// TIA Portal V21 export
DATA_BLOCK "RMAdd"   // DB305
AUTHOR : PRECISE
FAMILY : PRECISE
// stored: AutoNumber false, InstanceOfName FB310, InstanceOfType FB
"FB310"
   // VAR_INPUT
   //    Enable : Bool;
   //    Disable : Bool;
   //    Fault : Bool;
   //    SecPulse : Bool;
   //    AlwaysTrue : Bool;
   //    StartConfirmationPopupSel : Bool;
   //    EndConfirmationPopupSel : Bool;
   //    RMAddTypeSel : Int;   // RMAddTypeSel: 0-Manual/1-LIst MAnual
   //    RMTypeSel : Int;
   //    WeightBasedSel : Bool;
   //    AdditionMethodSel : Bool;
   //    RMAddPopupSel : Bool;
   //    SetRMNo : Int;
   //    "SetVacuum/SetPressure" : Real;
   //    SetQuantity : Real;
   //    SetSpeed : Real;
   //    "ActualVacuum/ActualPressure" : Real;
   //    ActualQuantity : Real;
   //    ActualQuantityRMVessel : Real;
   //    "VacuumTol/PressureTol" : Real;
   //    DelaytoSettleMaterial : Int;
   //    InflightQuantitySuction : Real;
   //    InflightQuantityLiqDrum : Real;
   //    DelaytoStartPump : Int;
   // END_VAR
   // VAR_OUTPUT
   //    VacuumInValve : Bool;
   //    VacuumLineValves : Bool;
   //    SuctionInValve : Bool;
   //    VacuumPumpCmd : Bool;
   //    LineValves : Bool;
   //    PumpCmd : Bool;
   //    StartConfirmationPopup : Bool;
   //    EndConfirmationPopup : Bool;
   //    DelaytoSettleMaterialPopup : Bool;
   //    RMAddPopup : Bool;
   //    RMAddPopupManual : Bool;
   //    ActualSpeed : Real;
   //    VisibleRM1 : Bool;
   //    VisibleRM2 : Bool;
   //    VisibleRM3 : Bool;
   //    VisibleRM4 : Bool;
   //    VisibleRM5 : Bool;
   //    VisibleRM6 : Bool;
   //    VisibleRM7 : Bool;
   //    VisibleRM8 : Bool;
   //    VisibleRM9 : Bool;
   //    VisibleRM10 : Bool;
   //    PrintTrigger : Bool;
   //    PrintWord : Int;
   //    PrintStatus : String[50];
   // END_VAR
   // VAR_IN_OUT
   //    Start : Bool;
   //    Stop : Bool;
   //    Reset : Bool;
   //    StartConfirmationAck : Bool;
   //    EndConfirmationAck : Bool;
   //    SpareBtn1 : Bool;
   //    SpareBtn2 : Bool;
   //    Running : Bool;
   //    Selected : Bool;
   //    Paused : Bool;
   //    StartConfirmationPopupTemp : Bool;
   //    EndConfirmationPopupTemp : Bool;
   //    RMAddPopupTemp : Bool;
   //    RMAddStarted : Bool;
   //    RMAddOver : Bool;
   //    ActualSetQuantityCalc : Real;
   //    ActualSetQuantity : Real;
   //    RMAddAck1 : Bool;
   //    RMAddAck2 : Bool;
   //    RMAddAck3 : Bool;
   //    RMAddAck4 : Bool;
   //    RMAddAck5 : Bool;
   //    RMAddAck6 : Bool;
   //    RMAddAck7 : Bool;
   //    RMAddAck8 : Bool;
   //    RMAddAck9 : Bool;
   //    RMAddAck10 : Bool;
   // END_VAR
   // VAR
   //    PrintTriggerTemp : Bool;
   //    RE1 : Bool;
   //    RE2 : Bool;
   //    RE3 : Bool;
   //    RE4 : Bool;
   //    RE5 : Bool;
   //    RE6 : Bool;
   //    RE7 : Bool;
   //    RE8 : Bool;
   //    RE9 : Bool;
   //    RE10 : Bool;
   //    RE11 : Bool;
   //    PrintTriggerResetTimer { S7_SetPoint := 'True'} : TON_TIME;
   //    BtnResetTimer { S7_SetPoint := 'True'} : TON_TIME;
   // END_VAR
   // VAR RETAIN
   //    NameRM1 : String[100];
   // END_VAR
   // VAR
   //    NameRM2 : String[100];
   //    NameRM3 : String[100];
   //    NameRM4 : String[100];
   //    NameRM5 : String[100];
   //    NameRM6 : String[100];
   //    NameRM7 : String[100];
   //    NameRM8 : String[100];
   //    NameRM9 : String[100];
   //    NameRM10 : String[100];
   //    Manual { S7_SetPoint := 'True'} : "FB307";
   //    Suction { S7_SetPoint := 'True'} : "FB308";
   //    LiqDrum { S7_SetPoint := 'True'} : "FB309";
   // END_VAR
BEGIN
END_DATA_BLOCK
